# EPICS autosave request: iocBoot/sioc-diag0-fc01/sioc-diag0-fc01.req
file "lcls2farc.req" AREA=DIAG0,POS=530
